LIN {X 0,Y 108.668,Z 991.691,A -85,B 0,C 180,E1 6722.041,E2 6722.041} C_VEL
LIN {X 0,Y 115.964,Z 986.125,A -85,B 0,C 180,E1 6711.629,E2 6711.629} C_VEL
LIN {X 0,Y 125.828,Z 978.975,A -85,B 0,C 180,E1 6703.029,E2 6703.029} C_VEL
LIN {X 0,Y 137.396,Z 970.37,A -85,B 0,C 180,E1 6696.117,E2 6696.117} C_VEL
LIN {X 0,Y 150.62,Z 959.785,A -85,B 0,C 180,E1 6690.352,E2 6690.352} C_VEL
LIN {X 0,Y 164.355,Z 947.613,A -85,B 0,C 180,E1 6685.798,E2 6685.798} C_VEL
LIN {X 0,Y 178.144,Z 933.873,A -85,B 0,C 180,E1 6682.172,E2 6682.172} C_VEL
LIN {X 0,Y 191.294,Z 919.026,A -85,B 0,C 180,E1 6679.367,E2 6679.367} C_VEL
LIN {X 0,Y 203.581,Z 903.149,A -85,B 0,C 180,E1 6677.161,E2 6677.161} C_VEL
LIN {X 0,Y 214.716,Z 886.544,A -85,B 0,C 180,E1 6675.442,E2 6675.442} C_VEL
LIN {X 0,Y 224.723,Z 869.138,A -85,B 0,C 180,E1 6674.088,E2 6674.088} C_VEL
LIN {X 0,Y 233.483,Z 851.076,A -85,B 0,C 180,E1 6673.039,E2 6673.039} C_VEL
LIN {X 0,Y 241.401,Z 830.942,A -85,B 0,C 180,E1 6672.186,E2 6672.186} C_VEL
LIN {X 0,Y 247.582,Z 810.659,A -85,B 0,C 180,E1 6671.567,E2 6671.567} C_VEL
LIN {X 0,Y 252.1,Z 790.058,A -85,B 0,C 180,E1 6671.085,E2 6671.085} C_VEL
LIN {X 0,Y 255.437,Z 766.946,A -85,B 0,C 180,E1 6670.837,E2 6670.837} C_VEL
LIN {X 0,Y 255.799,Z 763.582,A -85,B 0,C 180,E1 6670.771,E2 6670.771} C_VEL
LIN {X 0,Y 256.748,Z 736.616,A -85,B 0,C 180,E1 6667.524,E2 6667.524} C_VEL
LIN {X 0,Y 258.923,Z 706.753,A -85,B 0,C 180,E1 6664.457,E2 6664.457} C_VEL
LIN {X 0,Y 259.843,Z 696.602,A -85,B 0,C 180,E1 6663.474,E2 6663.474} C_VEL
LIN {X 0,Y 260.238,Z 689.281,A -85,B 0,C 180,E1 6660.825,E2 6660.825} C_VEL
LIN {X 0,Y 262.188,Z 677.578,A -85,B 0,C 180,E1 6656.009,E2 6656.009} C_VEL
LIN {X 0,Y 264.904,Z 669.637,A -85,B 0,C 180,E1 6652.19,E2 6652.19} C_VEL
LIN {X 0,Y 265.193,Z 670.053,A -85,B 0,C 180,E1 6651.653,E2 6651.653} C_VEL
LIN {X 0,Y 265.852,Z 672.18,A -85,B 0,C 180,E1 6650.356,E2 6650.356} C_VEL
LIN {X 0,Y 253.789,Z 778.906,A -85,B 0,C 180,E1 6648.472,E2 6648.472} C_VEL
LIN {X 0,Y 249.847,Z 799.249,A -85,B 0,C 180,E1 6647.946,E2 6647.946} C_VEL
LIN {X 0,Y 244.412,Z 819.077,A -85,B 0,C 180,E1 6647.237,E2 6647.237} C_VEL
LIN {X 0,Y 237.235,Z 839.076,A -85,B 0,C 180,E1 6646.276,E2 6646.276} C_VEL
LIN {X 0,Y 229.134,Z 857.25,A -85,B 0,C 180,E1 6645.133,E2 6645.133} C_VEL
LIN {X 0,Y 219.778,Z 874.734,A -85,B 0,C 180,E1 6643.719,E2 6643.719} C_VEL
LIN {X 0,Y 208.758,Z 892.029,A -85,B 0,C 180,E1 6641.89,E2 6641.89} C_VEL
LIN {X 0,Y 197.188,Z 907.581,A -85,B 0,C 180,E1 6639.724,E2 6639.724} C_VEL
LIN {X 0,Y 184.631,Z 922.268,A -85,B 0,C 180,E1 6637.014,E2 6637.014} C_VEL
LIN {X 0,Y 171.721,Z 935.505,A -85,B 0,C 180,E1 6633.721,E2 6633.721} C_VEL
LIN {X 0,Y 158.692,Z 947.341,A -85,B 0,C 180,E1 6629.672,E2 6629.672} C_VEL
LIN {X 0,Y 145.849,Z 957.776,A -85,B 0,C 180,E1 6624.663,E2 6624.663} C_VEL
LIN {X 0,Y 133.035,Z 967.156,A -85,B 0,C 180,E1 6618.075,E2 6618.075} C_VEL
LIN {X 0,Y 121.672,Z 974.814,A -85,B 0,C 180,E1 6609.862,E2 6609.862} C_VEL
LIN {X 0,Y 112.966,Z 980.439,A -85,B 0,C 180,E1 6600.295,E2 6600.295} C_VEL
LIN {X 0,Y 107.484,Z 984.062,A -85,B 0,C 180,E1 6590.023,E2 6590.023} C_VEL
LIN {X 0,Y 104.893,Z 986.058,A -85,B 0,C 180,E1 6579.323,E2 6579.323} C_VEL
LIN {X 0,Y 104.395,Z 986.656,A -85,B 0,C 180,E1 6569.997,E2 6569.997} C_VEL
LIN {X 0,Y 104.885,Z 986.083,A -85,B 0,C 180,E1 6560.671,E2 6560.671} C_VEL
LIN {X 0,Y 107.419,Z 984.152,A -85,B 0,C 180,E1 6550.072,E2 6550.072} C_VEL
LIN {X 0,Y 112.922,Z 980.53,A -85,B 0,C 180,E1 6539.685,E2 6539.685} C_VEL
LIN {X 0,Y 121.613,Z 974.922,A -85,B 0,C 180,E1 6530.109,E2 6530.109} C_VEL
LIN {X 0,Y 132.383,Z 967.681,A -85,B 0,C 180,E1 6522.238,E2 6522.238} C_VEL
LIN {X 0,Y 144.419,Z 958.957,A -85,B 0,C 180,E1 6515.898,E2 6515.898} C_VEL
LIN {X 0,Y 157.325,Z 948.621,A -85,B 0,C 180,E1 6510.697,E2 6510.697} C_VEL
LIN {X 0,Y 147.051,Z 951.529,A -85,B 0,C 180,E1 6506.23,E2 6506.23} C_VEL
LIN {X 0,Y 136.461,Z 954.568,A -85,B 0,C 180,E1 6499.698,E2 6499.698} C_VEL
LIN {X 0,Y 128.082,Z 957.332,A -85,B 0,C 180,E1 6491.711,E2 6491.711} C_VEL
LIN {X 0,Y 122.949,Z 959.82,A -85,B 0,C 180,E1 6483.264,E2 6483.264} C_VEL
LIN {X 0,Y 120.93,Z 962.742,A -85,B 0,C 180,E1 6471.921,E2 6471.921} C_VEL
LIN {X 0,Y 125.352,Z 965.819,A -85,B 0,C 180,E1 6458.475,E2 6458.475} C_VEL
LIN {X 0,Y 139.784,Z 968.622,A -85,B 0,C 180,E1 6445.025,E2 6445.025} C_VEL
LIN {X 0,Y 127.566,Z 977.809,A -85,B 0,C 180,E1 6438.129,E2 6438.129} C_VEL
LIN {X 0,Y 117.313,Z 985.24,A -85,B 0,C 180,E1 6429.738,E2 6429.738} C_VEL
LIN {X 0,Y 109.807,Z 990.867,A -85,B 0,C 180,E1 6420.021,E2 6420.021} C_VEL
LIN {X 0,Y 106.896,Z 992.481,A -85,B 0,C 180,E1 6416.302,E2 6416.302} C_VEL
LIN {X 0,Y 97.532,Z 995.483,A -85,B 0,C 180,E1 6405.695,E2 6405.695} C_VEL
LIN {X 0,Y 96.381,Z 996.081,A -85,B 0,C 180,E1 6401.813,E2 6401.813} C_VEL
LIN {X 0,Y 96.466,Z 996.89,A -85,B 0,C 180,E1 6392.974,E2 6392.974} C_VEL
LIN {X 0,Y 96.487,Z 996.912,A -85,B 0,C 180,E1 6387.628,E2 6387.628} C_VEL
LIN {X 0,Y 96.343,Z 996.122,A -85,B 0,C 180,E1 6378.631,E2 6378.631} C_VEL
LIN {X 0,Y 98.527,Z 993.582,A -85,B 0,C 180,E1 6366.689,E2 6366.689} C_VEL
LIN {X 0,Y 104.163,Z 989.385,A -85,B 0,C 180,E1 6355.508,E2 6355.508} C_VEL
LIN {X 0,Y 113.072,Z 983.454,A -85,B 0,C 180,E1 6345.691,E2 6345.691} C_VEL
LIN {X 0,Y 124.689,Z 975.635,A -85,B 0,C 180,E1 6337.456,E2 6337.456} C_VEL
LIN {X 0,Y 137.668,Z 966.274,A -85,B 0,C 180,E1 6331.021,E2 6331.021} C_VEL
LIN {X 0,Y 151.3,Z 955.493,A -85,B 0,C 180,E1 6326.01,E2 6326.01} C_VEL
LIN {X 0,Y 165.287,Z 943.149,A -85,B 0,C 180,E1 6322.027,E2 6322.027} C_VEL
LIN {X 0,Y 179.539,Z 928.903,A -85,B 0,C 180,E1 6318.79,E2 6318.79} C_VEL
LIN {X 0,Y 192.745,Z 913.813,A -85,B 0,C 180,E1 6316.331,E2 6316.331} C_VEL
LIN {X 0,Y 205.021,Z 897.675,A -85,B 0,C 180,E1 6314.401,E2 6314.401} C_VEL
LIN {X 0,Y 216.392,Z 880.245,A -85,B 0,C 180,E1 6312.859,E2 6312.859} C_VEL
LIN {X 0,Y 226.628,Z 861.559,A -85,B 0,C 180,E1 6311.646,E2 6311.646} C_VEL
LIN {X 0,Y 235.094,Z 842.869,A -85,B 0,C 180,E1 6310.758,E2 6310.758} C_VEL
LIN {X 0,Y 242.203,Z 823.431,A -85,B 0,C 180,E1 6310.085,E2 6310.085} C_VEL
LIN {X 0,Y 248.112,Z 802.126,A -85,B 0,C 180,E1 6309.543,E2 6309.543} C_VEL
LIN {X 0,Y 252.098,Z 781.253,A -85,B 0,C 180,E1 6309.166,E2 6309.166} C_VEL
LIN {X 0,Y 254.15,Z 765.555,A -85,B 0,C 180,E1 6309.011,E2 6309.011} C_VEL
LIN {X 0,Y 255.491,Z 739.464,A -85,B 0,C 180,E1 6305.868,E2 6305.868} C_VEL
LIN {X 0,Y 258.115,Z 709.106,A -85,B 0,C 180,E1 6302.761,E2 6302.761} C_VEL
LIN {X 0,Y 258.855,Z 701.864,A -85,B 0,C 180,E1 6302.047,E2 6302.047} C_VEL
LIN {X 0,Y 259.505,Z 694.909,A -85,B 0,C 180,E1 6299.448,E2 6299.448} C_VEL
LIN {X 0,Y 261.599,Z 684.612,A -85,B 0,C 180,E1 6295.176,E2 6295.176} C_VEL
LIN {X 0,Y 264.006,Z 677.964,A -85,B 0,C 180,E1 6291.973,E2 6291.973} C_VEL
LIN {X 0,Y 252.295,Z 779.354,A -85,B 0,C 180,E1 6290.249,E2 6290.249} C_VEL
LIN {X 0,Y 248.269,Z 799.753,A -85,B 0,C 180,E1 6289.747,E2 6289.747} C_VEL
LIN {X 0,Y 242.759,Z 819.493,A -85,B 0,C 180,E1 6289.078,E2 6289.078} C_VEL
LIN {X 0,Y 235.463,Z 839.469,A -85,B 0,C 180,E1 6288.17,E2 6288.17} C_VEL
LIN {X 0,Y 227.208,Z 857.649,A -85,B 0,C 180,E1 6287.088,E2 6287.088} C_VEL
LIN {X 0,Y 217.663,Z 875.137,A -85,B 0,C 180,E1 6285.749,E2 6285.749} C_VEL
LIN {X 0,Y 206.443,Z 892.371,A -85,B 0,C 180,E1 6284.021,E2 6284.021} C_VEL
LIN {X 0,Y 194.54,Z 907.991,A -85,B 0,C 180,E1 6281.952,E2 6281.952} C_VEL
LIN {X 0,Y 181.629,Z 922.681,A -85,B 0,C 180,E1 6279.36,E2 6279.36} C_VEL
LIN {X 0,Y 168.111,Z 936.089,A -85,B 0,C 180,E1 6276.143,E2 6276.143} C_VEL
LIN {X 0,Y 154.756,Z 947.757,A -85,B 0,C 180,E1 6272.265,E2 6272.265} C_VEL
LIN {X 0,Y 141.31,Z 958.194,A -85,B 0,C 180,E1 6267.348,E2 6267.348} C_VEL
LIN {X 0,Y 127.75,Z 967.574,A -85,B 0,C 180,E1 6260.787,E2 6260.787} C_VEL
LIN {X 0,Y 116.08,Z 974.902,A -85,B 0,C 180,E1 6252.877,E2 6252.877} C_VEL
LIN {X 0,Y 106.817,Z 980.371,A -85,B 0,C 180,E1 6243.519,E2 6243.519} C_VEL
LIN {X 0,Y 100.443,Z 984.148,A -85,B 0,C 180,E1 6232.841,E2 6232.841} C_VEL
LIN {X 0,Y 97.156,Z 986.346,A -85,B 0,C 180,E1 6221.273,E2 6221.273} C_VEL
LIN {X 0,Y 96.405,Z 987.005,A -85,B 0,C 180,E1 6211.78,E2 6211.78} C_VEL
LIN {X 0,Y 96.706,Z 986.749,A -85,B 0,C 180,E1 6202.272,E2 6202.272} C_VEL
LIN {X 0,Y 98.745,Z 985.269,A -85,B 0,C 180,E1 6191.703,E2 6191.703} C_VEL
LIN {X 0,Y 103.864,Z 982.144,A -85,B 0,C 180,E1 6180.593,E2 6180.593} C_VEL
LIN {X 0,Y 112.481,Z 977.086,A -85,B 0,C 180,E1 6170.204,E2 6170.204} C_VEL
LIN {X 0,Y 123.359,Z 970.453,A -85,B 0,C 180,E1 6161.778,E2 6161.778} C_VEL
LIN {X 0,Y 135.623,Z 962.37,A -85,B 0,C 180,E1 6155.078,E2 6155.078} C_VEL
LIN {X 0,Y 146.77,Z 954.193,A -85,B 0,C 180,E1 6150.387,E2 6150.387} C_VEL
LIN {X 0,Y 130.806,Z 958.339,A -85,B 0,C 180,E1 6141.526,E2 6141.526} C_VEL
LIN {X 0,Y 121.494,Z 961.15,A -85,B 0,C 180,E1 6132.839,E2 6132.839} C_VEL
LIN {X 0,Y 116.002,Z 963.516,A -85,B 0,C 180,E1 6123.955,E2 6123.955} C_VEL
LIN {X 0,Y 113.721,Z 966.225,A -85,B 0,C 180,E1 6112.422,E2 6112.422} C_VEL
LIN {X 0,Y 118.395,Z 969.376,A -85,B 0,C 180,E1 6097.665,E2 6097.665} C_VEL
LIN {X 0,Y 130.332,Z 971.766,A -85,B 0,C 180,E1 6085.562,E2 6085.562} C_VEL
LIN {X 0,Y 118.034,Z 980.243,A -85,B 0,C 180,E1 6078.201,E2 6078.201} C_VEL
LIN {X 0,Y 107.403,Z 987.311,A -85,B 0,C 180,E1 6068.593,E2 6068.593} C_VEL
LIN {X 0,Y 100.103,Z 992.425,A -85,B 0,C 180,E1 6057.259,E2 6057.259} C_VEL
LIN {X 0,Y 96.753,Z 995.452,A -85,B 0,C 180,E1 6045.59,E2 6045.59} C_VEL
LIN {X 0,Y 96.381,Z 996.081,A -85,B 0,C 180,E1 6041.813,E2 6041.813} C_VEL
LIN {X 0,Y 95.319,Z 996.58,A -85,B 0,C 180,E1 6037.558,E2 6037.558} C_VEL
LIN {X 0,Y 92.506,Z 996.742,A -85,B 0,C 180,E1 6032.007,E2 6032.007} C_VEL
LIN {X 0,Y 88.396,Z 996.199,A -85,B 0,C 180,E1 6021.798,E2 6021.798} C_VEL
LIN {X 0,Y 88.298,Z 995.978,A -85,B 0,C 180,E1 6019.947,E2 6019.947} C_VEL
LIN {X 0,Y 90.039,Z 994.007,A -85,B 0,C 180,E1 6007.821,E2 6007.821} C_VEL
LIN {X 0,Y 95.911,Z 989.964,A -85,B 0,C 180,E1 5995.019,E2 5995.019} C_VEL
LIN {X 0,Y 105.121,Z 984.331,A -85,B 0,C 180,E1 5984.495,E2 5984.495} C_VEL
LIN {X 0,Y 117.166,Z 976.876,A -85,B 0,C 180,E1 5975.84,E2 5975.84} C_VEL
LIN {X 0,Y 131.337,Z 967.426,A -85,B 0,C 180,E1 5968.902,E2 5968.902} C_VEL
LIN {X 0,Y 146.246,Z 956.361,A -85,B 0,C 180,E1 5963.638,E2 5963.638} C_VEL
LIN {X 0,Y 160.46,Z 944.482,A -85,B 0,C 180,E1 5959.801,E2 5959.801} C_VEL
LIN {X 0,Y 174.409,Z 931.286,A -85,B 0,C 180,E1 5956.793,E2 5956.793} C_VEL
LIN {X 0,Y 188.338,Z 916.157,A -85,B 0,C 180,E1 5954.342,E2 5954.342} C_VEL
LIN {X 0,Y 201.277,Z 899.839,A -85,B 0,C 180,E1 5952.434,E2 5952.434} C_VEL
LIN {X 0,Y 212.854,Z 882.789,A -85,B 0,C 180,E1 5950.969,E2 5950.969} C_VEL
LIN {X 0,Y 223.238,Z 864.744,A -85,B 0,C 180,E1 5949.825,E2 5949.825} C_VEL
LIN {X 0,Y 232.29,Z 845.836,A -85,B 0,C 180,E1 5948.949,E2 5948.949} C_VEL
LIN {X 0,Y 239.724,Z 826.696,A -85,B 0,C 180,E1 5948.303,E2 5948.303} C_VEL
LIN {X 0,Y 245.869,Z 806.184,A -85,B 0,C 180,E1 5947.797,E2 5947.797} C_VEL
LIN {X 0,Y 250.344,Z 784.986,A -85,B 0,C 180,E1 5947.404,E2 5947.404} C_VEL
LIN {X 0,Y 252.729,Z 767.652,A -85,B 0,C 180,E1 5947.23,E2 5947.23} C_VEL
LIN {X 0,Y 254.698,Z 739.448,A -85,B 0,C 180,E1 5943.883,E2 5943.883} C_VEL
LIN {X 0,Y 257.88,Z 708.454,A -85,B 0,C 180,E1 5940.777,E2 5940.777} C_VEL
LIN {X 0,Y 258.046,Z 706.967,A -85,B 0,C 180,E1 5940.555,E2 5940.555} C_VEL
LIN {X 0,Y 260.917,Z 692.086,A -85,B 0,C 180,E1 5934.557,E2 5934.557} C_VEL
LIN {X 0,Y 261.634,Z 690.138,A -85,B 0,C 180,E1 5933.511,E2 5933.511} C_VEL
LIN {X 0,Y 251.012,Z 780.054,A -85,B 0,C 180,E1 5932.04,E2 5932.04} C_VEL
LIN {X 0,Y 246.912,Z 800.368,A -85,B 0,C 180,E1 5931.566,E2 5931.566} C_VEL
LIN {X 0,Y 241.363,Z 819.898,A -85,B 0,C 180,E1 5930.943,E2 5930.943} C_VEL
LIN {X 0,Y 233.952,Z 839.861,A -85,B 0,C 180,E1 5930.091,E2 5930.091} C_VEL
LIN {X 0,Y 225.552,Z 858.049,A -85,B 0,C 180,E1 5929.074,E2 5929.074} C_VEL
LIN {X 0,Y 215.826,Z 875.541,A -85,B 0,C 180,E1 5927.817,E2 5927.817} C_VEL
LIN {X 0,Y 204.374,Z 892.778,A -85,B 0,C 180,E1 5926.19,E2 5926.19} C_VEL
LIN {X 0,Y 192.195,Z 908.402,A -85,B 0,C 180,E1 5924.238,E2 5924.238} C_VEL
LIN {X 0,Y 178.942,Z 923.093,A -85,B 0,C 180,E1 5921.781,E2 5921.781} C_VEL
LIN {X 0,Y 164.677,Z 936.795,A -85,B 0,C 180,E1 5918.635,E2 5918.635} C_VEL
LIN {X 0,Y 150.348,Z 948.793,A -85,B 0,C 180,E1 5914.743,E2 5914.743} C_VEL
LIN {X 0,Y 136.348,Z 959.111,A -85,B 0,C 180,E1 5909.913,E2 5909.913} C_VEL
LIN {X 0,Y 122.776,Z 967.992,A -85,B 0,C 180,E1 5903.725,E2 5903.725} C_VEL
LIN {X 0,Y 109.702,Z 975.651,A -85,B 0,C 180,E1 5895.306,E2 5895.306} C_VEL
LIN {X 0,Y 99.305,Z 981.275,A -85,B 0,C 180,E1 5885.019,E2 5885.019} C_VEL
LIN {X 0,Y 92.523,Z 984.866,A -85,B 0,C 180,E1 5873.565,E2 5873.565} C_VEL
LIN {X 0,Y 89.095,Z 986.885,A -85,B 0,C 180,E1 5860.995,E2 5860.995} C_VEL
LIN {X 0,Y 88.415,Z 987.479,A -85,B 0,C 180,E1 5849.997,E2 5849.997} C_VEL
LIN {X 0,Y 89.086,Z 986.91,A -85,B 0,C 180,E1 5838.997,E2 5838.997} C_VEL
LIN {X 0,Y 92.247,Z 985.074,A -85,B 0,C 180,E1 5827.029,E2 5827.029} C_VEL
LIN {X 0,Y 99.263,Z 981.362,A -85,B 0,C 180,E1 5814.956,E2 5814.956} C_VEL
LIN {X 0,Y 109.851,Z 975.646,A -85,B 0,C 180,E1 5804.496,E2 5804.496} C_VEL
LIN {X 0,Y 122.715,Z 968.129,A -85,B 0,C 180,E1 5796.227,E2 5796.227} C_VEL
LIN {X 0,Y 136.43,Z 959.178,A -85,B 0,C 180,E1 5789.952,E2 5789.952} C_VEL
LIN {X 0,Y 124.656,Z 961.988,A -85,B 0,C 180,E1 5783.144,E2 5783.144} C_VEL
LIN {X 0,Y 115.183,Z 964.621,A -85,B 0,C 180,E1 5774.581,E2 5774.581} C_VEL
LIN {X 0,Y 108.981,Z 967.029,A -85,B 0,C 180,E1 5764.737,E2 5764.737} C_VEL
LIN {X 0,Y 106.47,Z 969.602,A -85,B 0,C 180,E1 5752.446,E2 5752.446} C_VEL
LIN {X 0,Y 111.332,Z 972.629,A -85,B 0,C 180,E1 5736.725,E2 5736.725} C_VEL
LIN {X 0,Y 121.009,Z 974.573,A -85,B 0,C 180,E1 5726.251,E2 5726.251} C_VEL
LIN {X 0,Y 108.504,Z 982.374,A -85,B 0,C 180,E1 5718.285,E2 5718.285} C_VEL
LIN {X 0,Y 98.359,Z 988.484,A -85,B 0,C 180,E1 5708.326,E2 5708.326} C_VEL
LIN {X 0,Y 91.323,Z 993.026,A -85,B 0,C 180,E1 5695.976,E2 5695.976} C_VEL
LIN {X 0,Y 88.467,Z 995.643,A -85,B 0,C 180,E1 5683.068,E2 5683.068} C_VEL
LIN {X 0,Y 88.459,Z 996.477,A -85,B 0,C 180,E1 5673.243,E2 5673.243} C_VEL
LIN {X 0,Y 88.484,Z 996.499,A -85,B 0,C 180,E1 5667.413,E2 5667.413} C_VEL
LIN {X 0,Y 88.298,Z 995.978,A -85,B 0,C 180,E1 5659.947,E2 5659.947} C_VEL
LIN {X 0,Y 87.663,Z 995.347,A -85,B 0,C 180,E1 5654.929,E2 5654.929} C_VEL
LIN {X 0,Y 85.123,Z 993.386,A -85,B 0,C 180,E1 5644.717,E2 5644.717} C_VEL
LIN {X 0,Y 85.592,Z 991.753,A -85,B 0,C 180,E1 5638.425,E2 5638.425} C_VEL
LIN {X 0,Y 86.354,Z 991.183,A -85,B 0,C 180,E1 5636.672,E2 5636.672} C_VEL
LIN {X 0,Y 95.582,Z 986.11,A -85,B 0,C 180,E1 5624.661,E2 5624.661} C_VEL
LIN {X 0,Y 108.387,Z 978.945,A -85,B 0,C 180,E1 5614.818,E2 5614.818} C_VEL
LIN {X 0,Y 122.882,Z 970.112,A -85,B 0,C 180,E1 5607.518,E2 5607.518} C_VEL
LIN {X 0,Y 137.941,Z 959.823,A -85,B 0,C 180,E1 5602.142,E2 5602.142} C_VEL
LIN {X 0,Y 152.606,Z 948.48,A -85,B 0,C 180,E1 5598.197,E2 5598.197} C_VEL
LIN {X 0,Y 167.691,Z 935.177,A -85,B 0,C 180,E1 5595.006,E2 5595.006} C_VEL
LIN {X 0,Y 182.315,Z 920.329,A -85,B 0,C 180,E1 5592.535,E2 5592.535} C_VEL
LIN {X 0,Y 195.365,Z 905.022,A -85,B 0,C 180,E1 5590.7,E2 5590.7} C_VEL
LIN {X 0,Y 207.655,Z 888.259,A -85,B 0,C 180,E1 5589.231,E2 5589.231} C_VEL
LIN {X 0,Y 218.642,Z 870.536,A -85,B 0,C 180,E1 5588.093,E2 5588.093} C_VEL
LIN {X 0,Y 228.273,Z 851.881,A -85,B 0,C 180,E1 5587.221,E2 5587.221} C_VEL
LIN {X 0,Y 236.024,Z 833.581,A -85,B 0,C 180,E1 5586.596,E2 5586.596} C_VEL
LIN {X 0,Y 243.044,Z 812.513,A -85,B 0,C 180,E1 5586.075,E2 5586.075} C_VEL
LIN {X 0,Y 248.142,Z 791.369,A -85,B 0,C 180,E1 5585.668,E2 5585.668} C_VEL
LIN {X 0,Y 251.43,Z 770.926,A -85,B 0,C 180,E1 5585.483,E2 5585.483} C_VEL
LIN {X 0,Y 251.609,Z 768.944,A -85,B 0,C 180,E1 5585.329,E2 5585.329} C_VEL
LIN {X 0,Y 254.288,Z 738.743,A -85,B 0,C 180,E1 5581.83,E2 5581.83} C_VEL
LIN {X 0,Y 257.365,Z 712.416,A -85,B 0,C 180,E1 5579.165,E2 5579.165} C_VEL
LIN {X 0,Y 259.438,Z 702.446,A -85,B 0,C 180,E1 5575.073,E2 5575.073} C_VEL
LIN {X 0,Y 249.998,Z 780.612,A -85,B 0,C 180,E1 5573.851,E2 5573.851} C_VEL
LIN {X 0,Y 245.807,Z 800.988,A -85,B 0,C 180,E1 5573.403,E2 5573.403} C_VEL
LIN {X 0,Y 240.225,Z 820.305,A -85,B 0,C 180,E1 5572.827,E2 5572.827} C_VEL
LIN {X 0,Y 232.708,Z 840.253,A -85,B 0,C 180,E1 5572.034,E2 5572.034} C_VEL
LIN {X 0,Y 224.17,Z 858.447,A -85,B 0,C 180,E1 5571.087,E2 5571.087} C_VEL
LIN {X 0,Y 214.275,Z 875.944,A -85,B 0,C 180,E1 5569.917,E2 5569.917} C_VEL
LIN {X 0,Y 202.604,Z 893.185,A -85,B 0,C 180,E1 5568.401,E2 5568.401} C_VEL
LIN {X 0,Y 190.163,Z 908.811,A -85,B 0,C 180,E1 5566.577,E2 5566.577} C_VEL
LIN {X 0,Y 176.583,Z 923.506,A -85,B 0,C 180,E1 5564.27,E2 5564.27} C_VEL
LIN {X 0,Y 162.439,Z 936.748,A -85,B 0,C 180,E1 5561.421,E2 5561.421} C_VEL
LIN {X 0,Y 147.907,Z 948.59,A -85,B 0,C 180,E1 5557.833,E2 5557.833} C_VEL
LIN {X 0,Y 133.256,Z 959.028,A -85,B 0,C 180,E1 5553.234,E2 5553.234} C_VEL
LIN {X 0,Y 118.152,Z 968.41,A -85,B 0,C 180,E1 5546.902,E2 5546.902} C_VEL
LIN {X 0,Y 104.15,Z 976.069,A -85,B 0,C 180,E1 5538.483,E2 5538.483} C_VEL
LIN {X 0,Y 92.782,Z 981.693,A -85,B 0,C 180,E1 5527.894,E2 5527.894} C_VEL
LIN {X 0,Y 85.179,Z 985.282,A -85,B 0,C 180,E1 5515.738,E2 5515.738} C_VEL
LIN {X 0,Y 81.228,Z 987.299,A -85,B 0,C 180,E1 5502.075,E2 5502.075} C_VEL
LIN {X 0,Y 80.425,Z 987.89,A -85,B 0,C 180,E1 5489.996,E2 5489.996} C_VEL
LIN {X 0,Y 81.22,Z 987.323,A -85,B 0,C 180,E1 5477.916,E2 5477.916} C_VEL
LIN {X 0,Y 84.868,Z 985.49,A -85,B 0,C 180,E1 5464.9,E2 5464.9} C_VEL
LIN {X 0,Y 92.74,Z 981.779,A -85,B 0,C 180,E1 5452.078,E2 5452.078} C_VEL
LIN {X 0,Y 104.097,Z 976.172,A -85,B 0,C 180,E1 5441.475,E2 5441.475} C_VEL
LIN {X 0,Y 117.379,Z 968.936,A -85,B 0,C 180,E1 5433.402,E2 5433.402} C_VEL
LIN {X 0,Y 125.897,Z 963.88,A -85,B 0,C 180,E1 5429.499,E2 5429.499} C_VEL
LIN {X 0,Y 109.281,Z 967.732,A -85,B 0,C 180,E1 5417.025,E2 5417.025} C_VEL
LIN {X 0,Y 101.86,Z 970.281,A -85,B 0,C 180,E1 5405.634,E2 5405.634} C_VEL
LIN {X 0,Y 99.133,Z 972.793,A -85,B 0,C 180,E1 5392.467,E2 5392.467} C_VEL
LIN {X 0,Y 104.22,Z 975.673,A -85,B 0,C 180,E1 5375.637,E2 5375.637} C_VEL
LIN {X 0,Y 111.613,Z 977.111,A -85,B 0,C 180,E1 5367.02,E2 5367.02} C_VEL
LIN {X 0,Y 98.372,Z 984.613,A -85,B 0,C 180,E1 5357.87,E2 5357.87} C_VEL
LIN {X 0,Y 88.09,Z 990.241,A -85,B 0,C 180,E1 5346.177,E2 5346.177} C_VEL
LIN {X 0,Y 82.136,Z 993.87,A -85,B 0,C 180,E1 5332.93,E2 5332.93} C_VEL
LIN {X 0,Y 80.308,Z 995.761,A -85,B 0,C 180,E1 5319.318,E2 5319.318} C_VEL
LIN {X 0,Y 80.588,Z 996.183,A -85,B 0,C 180,E1 5310.004,E2 5310.004} C_VEL
LIN {X 0,Y 80.292,Z 995.745,A -85,B 0,C 180,E1 5300.687,E2 5300.687} C_VEL
LIN {X 0,Y 82.113,Z 993.843,A -85,B 0,C 180,E1 5287.071,E2 5287.071} C_VEL
LIN {X 0,Y 86.354,Z 991.183,A -85,B 0,C 180,E1 5276.672,E2 5276.672} C_VEL
LIN {X 0,Y 88.288,Z 989.594,A -85,B 0,C 180,E1 5271.849,E2 5271.849} C_VEL
LIN {X 0,Y 92.995,Z 984.521,A -85,B 0,C 180,E1 5259.103,E2 5259.103} C_VEL
LIN {X 0,Y 96.329,Z 982.492,A -85,B 0,C 180,E1 5255.831,E2 5255.831} C_VEL
LIN {X 0,Y 111.39,Z 974.362,A -85,B 0,C 180,E1 5247.303,E2 5247.303} C_VEL
LIN {X 0,Y 126.716,Z 965.004,A -85,B 0,C 180,E1 5241.402,E2 5241.402} C_VEL
LIN {X 0,Y 142.227,Z 954.227,A -85,B 0,C 180,E1 5237.051,E2 5237.051} C_VEL
LIN {X 0,Y 157.492,Z 942.084,A -85,B 0,C 180,E1 5233.759,E2 5233.759} C_VEL
LIN {X 0,Y 172.271,Z 928.585,A -85,B 0,C 180,E1 5231.233,E2 5231.233} C_VEL
LIN {X 0,Y 186.403,Z 913.679,A -85,B 0,C 180,E1 5229.26,E2 5229.26} C_VEL
LIN {X 0,Y 199.769,Z 897.261,A -85,B 0,C 180,E1 5227.702,E2 5227.702} C_VEL
LIN {X 0,Y 211.752,Z 879.886,A -85,B 0,C 180,E1 5226.507,E2 5226.507} C_VEL
LIN {X 0,Y 222.03,Z 862.147,A -85,B 0,C 180,E1 5225.618,E2 5225.618} C_VEL
LIN {X 0,Y 230.823,Z 843.924,A -85,B 0,C 180,E1 5224.951,E2 5224.951} C_VEL
LIN {X 0,Y 238.671,Z 823.735,A -85,B 0,C 180,E1 5224.421,E2 5224.421} C_VEL
LIN {X 0,Y 244.701,Z 803.397,A -85,B 0,C 180,E1 5224.024,E2 5224.024} C_VEL
LIN {X 0,Y 248.943,Z 783.329,A -85,B 0,C 180,E1 5223.732,E2 5223.732} C_VEL
LIN {X 0,Y 250.633,Z 771.769,A -85,B 0,C 180,E1 5223.616,E2 5223.616} C_VEL
LIN {X 0,Y 253.764,Z 741.686,A -85,B 0,C 180,E1 5220.155,E2 5220.155} C_VEL
LIN {X 0,Y 256.818,Z 718.012,A -85,B 0,C 180,E1 5217.768,E2 5217.768} C_VEL
LIN {X 0,Y 257.353,Z 715.466,A -85,B 0,C 180,E1 5216.651,E2 5216.651} C_VEL
LIN {X 0,Y 249.196,Z 781.427,A -85,B 0,C 180,E1 5215.67,E2 5215.67} C_VEL
LIN {X 0,Y 244.871,Z 801.964,A -85,B 0,C 180,E1 5215.246,E2 5215.246} C_VEL
LIN {X 0,Y 238.986,Z 821.798,A -85,B 0,C 180,E1 5214.691,E2 5214.691} C_VEL
LIN {X 0,Y 231.251,Z 841.752,A -85,B 0,C 180,E1 5213.948,E2 5213.948} C_VEL
LIN {X 0,Y 222.027,Z 860.761,A -85,B 0,C 180,E1 5213.016,E2 5213.016} C_VEL
LIN {X 0,Y 211.584,Z 878.522,A -85,B 0,C 180,E1 5211.885,E2 5211.885} C_VEL
LIN {X 0,Y 200.022,Z 895.097,A -85,B 0,C 180,E1 5210.505,E2 5210.505} C_VEL
LIN {X 0,Y 186.593,Z 911.396,A -85,B 0,C 180,E1 5208.689,E2 5208.689} C_VEL
LIN {X 0,Y 172.735,Z 925.732,A -85,B 0,C 180,E1 5206.512,E2 5206.512} C_VEL
LIN {X 0,Y 158.255,Z 938.669,A -85,B 0,C 180,E1 5203.803,E2 5203.803} C_VEL
LIN {X 0,Y 143.314,Z 950.245,A -85,B 0,C 180,E1 5200.359,E2 5200.359} C_VEL
LIN {X 0,Y 128.157,Z 960.446,A -85,B 0,C 180,E1 5195.891,E2 5195.891} C_VEL
LIN {X 0,Y 113.161,Z 969.22,A -85,B 0,C 180,E1 5189.98,E2 5189.98} C_VEL
LIN {X 0,Y 98.702,Z 976.603,A -85,B 0,C 180,E1 5181.833,E2 5181.833} C_VEL
LIN {X 0,Y 86.527,Z 982.111,A -85,B 0,C 180,E1 5171.193,E2 5171.193} C_VEL
LIN {X 0,Y 77.979,Z 985.699,A -85,B 0,C 180,E1 5158.317,E2 5158.317} C_VEL
LIN {X 0,Y 73.394,Z 987.712,A -85,B 0,C 180,E1 5143.387,E2 5143.387} C_VEL
LIN {X 0,Y 72.432,Z 988.283,A -85,B 0,C 180,E1 5130.787,E2 5130.787} C_VEL
LIN {X 0,Y 73.15,Z 987.861,A -85,B 0,C 180,E1 5118.164,E2 5118.164} C_VEL
LIN {X 0,Y 77.006,Z 986.195,A -85,B 0,C 180,E1 5103.799,E2 5103.799} C_VEL
LIN {X 0,Y 85.471,Z 982.609,A -85,B 0,C 180,E1 5089.949,E2 5089.949} C_VEL
LIN {X 0,Y 96.949,Z 977.462,A -85,B 0,C 180,E1 5079.327,E2 5079.327} C_VEL
LIN {X 0,Y 110.859,Z 970.526,A -85,B 0,C 180,E1 5071.033,E2 5071.033} C_VEL
LIN {X 0,Y 115.275,Z 968.146,A -85,B 0,C 180,E1 5068.893,E2 5068.893} C_VEL
LIN {X 0,Y 101.801,Z 971.069,A -85,B 0,C 180,E1 5057.727,E2 5057.727} C_VEL
LIN {X 0,Y 94.881,Z 973.189,A -85,B 0,C 180,E1 5047.266,E2 5047.266} C_VEL
LIN {X 0,Y 91.734,Z 975.802,A -85,B 0,C 180,E1 5031.855,E2 5031.855} C_VEL
LIN {X 0,Y 97.083,Z 978.526,A -85,B 0,C 180,E1 5014.371,E2 5014.371} C_VEL
LIN {X 0,Y 102.224,Z 979.477,A -85,B 0,C 180,E1 5007.924,E2 5007.924} C_VEL
LIN {X 0,Y 89.427,Z 986.042,A -85,B 0,C 180,E1 4998.518,E2 4998.518} C_VEL
LIN {X 0,Y 79.067,Z 991.127,A -85,B 0,C 180,E1 4985.575,E2 4985.575} C_VEL
LIN {X 0,Y 73.49,Z 994.194,A -85,B 0,C 180,E1 4970.721,E2 4970.721} C_VEL
LIN {X 0,Y 72.361,Z 995.584,A -85,B 0,C 180,E1 4955.821,E2 4955.821} C_VEL
LIN {X 0,Y 72.537,Z 995.726,A -85,B 0,C 180,E1 4948.424,E2 4948.424} C_VEL
LIN {X 0,Y 72.475,Z 995.021,A -85,B 0,C 180,E1 4936.44,E2 4936.44} C_VEL
LIN {X 0,Y 75.965,Z 992.656,A -85,B 0,C 180,E1 4920.861,E2 4920.861} C_VEL
LIN {X 0,Y 83.947,Z 988.644,A -85,B 0,C 180,E1 4907.247,E2 4907.247} C_VEL
LIN {X 0,Y 96.329,Z 982.492,A -85,B 0,C 180,E1 4895.831,E2 4895.831} C_VEL
LIN {X 0,Y 100.431,Z 979.975,A -85,B 0,C 180,E1 4892.284,E2 4892.284} C_VEL
LIN {X 0,Y 110.408,Z 972.731,A -85,B 0,C 180,E1 4882.87,E2 4882.87} C_VEL
LIN {X 0,Y 114.863,Z 969.999,A -85,B 0,C 180,E1 4880.749,E2 4880.749} C_VEL
LIN {X 0,Y 131.018,Z 960.023,A -85,B 0,C 180,E1 4875.945,E2 4875.945} C_VEL
LIN {X 0,Y 147.379,Z 948.347,A -85,B 0,C 180,E1 4872.339,E2 4872.339} C_VEL
LIN {X 0,Y 163.272,Z 935.193,A -85,B 0,C 180,E1 4869.628,E2 4869.628} C_VEL
LIN {X 0,Y 178.043,Z 921.027,A -85,B 0,C 180,E1 4867.623,E2 4867.623} C_VEL
LIN {X 0,Y 192.038,Z 905.416,A -85,B 0,C 180,E1 4866.052,E2 4866.052} C_VEL
LIN {X 0,Y 205.189,Z 888.161,A -85,B 0,C 180,E1 4864.811,E2 4864.811} C_VEL
LIN {X 0,Y 216.465,Z 870.536,A -85,B 0,C 180,E1 4863.899,E2 4863.899} C_VEL
LIN {X 0,Y 226.318,Z 852.083,A -85,B 0,C 180,E1 4863.209,E2 4863.209} C_VEL
LIN {X 0,Y 234.549,Z 833.244,A -85,B 0,C 180,E1 4862.703,E2 4862.703} C_VEL
LIN {X 0,Y 241.593,Z 812.72,A -85,B 0,C 180,E1 4862.305,E2 4862.305} C_VEL
LIN {X 0,Y 246.764,Z 792.244,A -85,B 0,C 180,E1 4861.982,E2 4861.982} C_VEL
LIN {X 0,Y 249.936,Z 773.78,A -85,B 0,C 180,E1 4861.791,E2 4861.791} C_VEL
LIN {X 0,Y 253.497,Z 744.346,A -85,B 0,C 180,E1 4858.446,E2 4858.446} C_VEL
LIN {X 0,Y 253.932,Z 741.148,A -85,B 0,C 180,E1 4858.079,E2 4858.079} C_VEL
LIN {X 0,Y 248.527,Z 782.97,A -85,B 0,C 180,E1 4857.486,E2 4857.486} C_VEL
LIN {X 0,Y 243.873,Z 804.255,A -85,B 0,C 180,E1 4857.071,E2 4857.071} C_VEL
LIN {X 0,Y 237.644,Z 824.351,A -85,B 0,C 180,E1 4856.541,E2 4856.541} C_VEL
LIN {X 0,Y 229.926,Z 843.547,A -85,B 0,C 180,E1 4855.873,E2 4855.873} C_VEL
LIN {X 0,Y 220.79,Z 861.896,A -85,B 0,C 180,E1 4855.04,E2 4855.04} C_VEL
LIN {X 0,Y 209.983,Z 879.846,A -85,B 0,C 180,E1 4853.986,E2 4853.986} C_VEL
LIN {X 0,Y 198.07,Z 896.477,A -85,B 0,C 180,E1 4852.704,E2 4852.704} C_VEL
LIN {X 0,Y 184.706,Z 912.322,A -85,B 0,C 180,E1 4851.074,E2 4851.074} C_VEL
LIN {X 0,Y 170.097,Z 927.052,A -85,B 0,C 180,E1 4848.998,E2 4848.998} C_VEL
LIN {X 0,Y 155.275,Z 939.836,A -85,B 0,C 180,E1 4846.483,E2 4846.483} C_VEL
LIN {X 0,Y 139.906,Z 951.28,A -85,B 0,C 180,E1 4843.259,E2 4843.259} C_VEL
LIN {X 0,Y 123.356,Z 961.863,A -85,B 0,C 180,E1 4838.762,E2 4838.762} C_VEL
LIN {X 0,Y 107.493,Z 970.54,A -85,B 0,C 180,E1 4832.884,E2 4832.884} C_VEL
LIN {X 0,Y 92.76,Z 977.492,A -85,B 0,C 180,E1 4825,E2 4825} C_VEL
LIN {X 0,Y 80.034,Z 982.759,A -85,B 0,C 180,E1 4814.39,E2 4814.39} C_VEL
LIN {X 0,Y 70.227,Z 986.416,A -85,B 0,C 180,E1 4799.883,E2 4799.883} C_VEL
LIN {X 0,Y 65.458,Z 988.188,A -85,B 0,C 180,E1 4784.141,E2 4784.141} C_VEL
LIN {X 0,Y 64.447,Z 988.713,A -85,B 0,C 180,E1 4769.995,E2 4769.995} C_VEL
LIN {X 0,Y 65.449,Z 988.212,A -85,B 0,C 180,E1 4755.847,E2 4755.847} C_VEL
LIN {X 0,Y 70.2,Z 986.471,A -85,B 0,C 180,E1 4740.094,E2 4740.094} C_VEL
LIN {X 0,Y 79.995,Z 982.83,A -85,B 0,C 180,E1 4725.572,E2 4725.572} C_VEL
LIN {X 0,Y 93.417,Z 977.296,A -85,B 0,C 180,E1 4714.493,E2 4714.493} C_VEL
LIN {X 0,Y 104.818,Z 971.972,A -85,B 0,C 180,E1 4708.208,E2 4708.208} C_VEL
LIN {X 0,Y 88.201,Z 975.823,A -85,B 0,C 180,E1 4689.791,E2 4689.791} C_VEL
LIN {X 0,Y 84.191,Z 978.467,A -85,B 0,C 180,E1 4671.808,E2 4671.808} C_VEL
LIN {X 0,Y 90.068,Z 981.147,A -85,B 0,C 180,E1 4652.641,E2 4652.641} C_VEL
LIN {X 0,Y 92.749,Z 981.666,A -85,B 0,C 180,E1 4648.947,E2 4648.947} C_VEL
LIN {X 0,Y 79.203,Z 987.783,A -85,B 0,C 180,E1 4638.006,E2 4638.006} C_VEL
LIN {X 0,Y 69.669,Z 991.933,A -85,B 0,C 180,E1 4624.041,E2 4624.041} C_VEL
LIN {X 0,Y 64.715,Z 994.542,A -85,B 0,C 180,E1 4606.152,E2 4606.152} C_VEL
LIN {X 0,Y 64.495,Z 995.292,A -85,B 0,C 180,E1 4592.67,E2 4592.67} C_VEL
LIN {X 0,Y 64.452,Z 995.26,A -85,B 0,C 180,E1 4586.447,E2 4586.447} C_VEL
LIN {X 0,Y 64.91,Z 994.369,A -85,B 0,C 180,E1 4572.062,E2 4572.062} C_VEL
LIN {X 0,Y 70.013,Z 991.722,A -85,B 0,C 180,E1 4555.168,E2 4555.168} C_VEL
LIN {X 0,Y 80.43,Z 987.157,A -85,B 0,C 180,E1 4540.69,E2 4540.69} C_VEL
LIN {X 0,Y 93.842,Z 981.024,A -85,B 0,C 180,E1 4530.347,E2 4530.347} C_VEL
LIN {X 0,Y 108.675,Z 973.49,A -85,B 0,C 180,E1 4523.074,E2 4523.074} C_VEL
LIN {X 0,Y 114.863,Z 969.999,A -85,B 0,C 180,E1 4520.749,E2 4520.749} C_VEL
LIN {X 0,Y 120.114,Z 966.747,A -85,B 0,C 180,E1 4518.451,E2 4518.451} C_VEL
LIN {X 0,Y 132.748,Z 957.368,A -85,B 0,C 180,E1 4511.989,E2 4511.989} C_VEL
LIN {X 0,Y 137.546,Z 953.906,A -85,B 0,C 180,E1 4510.676,E2 4510.676} C_VEL
LIN {X 0,Y 154.417,Z 941.244,A -85,B 0,C 180,E1 4507.841,E2 4507.841} C_VEL
LIN {X 0,Y 169.846,Z 927.75,A -85,B 0,C 180,E1 4505.82,E2 4505.82} C_VEL
LIN {X 0,Y 184.479,Z 912.856,A -85,B 0,C 180,E1 4504.263,E2 4504.263} C_VEL
LIN {X 0,Y 198.247,Z 896.44,A -85,B 0,C 180,E1 4503.048,E2 4503.048} C_VEL
LIN {X 0,Y 210.609,Z 878.96,A -85,B 0,C 180,E1 4502.121,E2 4502.121} C_VEL
LIN {X 0,Y 221.034,Z 861.344,A -85,B 0,C 180,E1 4501.451,E2 4501.451} C_VEL
LIN {X 0,Y 229.994,Z 843.137,A -85,B 0,C 180,E1 4500.951,E2 4500.951} C_VEL
LIN {X 0,Y 237.972,Z 822.969,A -85,B 0,C 180,E1 4500.561,E2 4500.561} C_VEL
LIN {X 0,Y 244.11,Z 802.627,A -85,B 0,C 180,E1 4500.259,E2 4500.259} C_VEL
LIN {X 0,Y 248.428,Z 782.583,A -85,B 0,C 180,E1 4500.042,E2 4500.042} C_VEL
LIN {X 0,Y 249.464,Z 775.759,A -85,B 0,C 180,E1 4499.957,E2 4499.957} C_VEL
LIN {X 0,Y 250.021,Z 772.054,A -85,B 0,C 180,E1 4499.488,E2 4499.488} C_VEL
LIN {X 0,Y 246.226,Z 793.811,A -85,B 0,C 180,E1 4499.159,E2 4499.159} C_VEL
LIN {X 0,Y 240.676,Z 814.671,A -85,B 0,C 180,E1 4498.729,E2 4498.729} C_VEL
LIN {X 0,Y 234.074,Z 833.181,A -85,B 0,C 180,E1 4498.223,E2 4498.223} C_VEL
LIN {X 0,Y 225.667,Z 851.975,A -85,B 0,C 180,E1 4497.561,E2 4497.561} C_VEL
LIN {X 0,Y 215.812,Z 869.99,A -85,B 0,C 180,E1 4496.745,E2 4496.745} C_VEL
LIN {X 0,Y 204.533,Z 887.194,A -85,B 0,C 180,E1 4495.732,E2 4495.732} C_VEL
LIN {X 0,Y 191.374,Z 904.04,A -85,B 0,C 180,E1 4494.421,E2 4494.421} C_VEL
LIN {X 0,Y 176.883,Z 919.692,A -85,B 0,C 180,E1 4492.753,E2 4492.753} C_VEL
LIN {X 0,Y 162.08,Z 933.302,A -85,B 0,C 180,E1 4490.749,E2 4490.749} C_VEL
LIN {X 0,Y 146.49,Z 945.603,A -85,B 0,C 180,E1 4488.184,E2 4488.184} C_VEL
LIN {X 0,Y 129.593,Z 956.981,A -85,B 0,C 180,E1 4484.662,E2 4484.662} C_VEL
LIN {X 0,Y 112.788,Z 966.573,A -85,B 0,C 180,E1 4479.99,E2 4479.99} C_VEL
LIN {X 0,Y 96.925,Z 974.27,A -85,B 0,C 180,E1 4473.82,E2 4473.82} C_VEL
LIN {X 0,Y 81.546,Z 980.602,A -85,B 0,C 180,E1 4464.809,E2 4464.809} C_VEL
LIN {X 0,Y 68.096,Z 985.326,A -85,B 0,C 180,E1 4451.35,E2 4451.35} C_VEL
LIN {X 0,Y 59.51,Z 988.045,A -85,B 0,C 180,E1 4433.775,E2 4433.775} C_VEL
LIN {X 0,Y 56.588,Z 989.002,A -85,B 0,C 180,E1 4416.08,E2 4416.08} C_VEL
LIN {X 0,Y 56.584,Z 989.01,A -85,B 0,C 180,E1 4403.908,E2 4403.908} C_VEL
LIN {X 0,Y 59.489,Z 988.084,A -85,B 0,C 180,E1 4386.205,E2 4386.205} C_VEL
LIN {X 0,Y 68.062,Z 985.384,A -85,B 0,C 180,E1 4368.613,E2 4368.613} C_VEL
LIN {X 0,Y 81.214,Z 980.782,A -85,B 0,C 180,E1 4355.356,E2 4355.356} C_VEL
LIN {X 0,Y 94.048,Z 975.572,A -85,B 0,C 180,E1 4347.379,E2 4347.379} C_VEL
LIN {X 0,Y 80.153,Z 978.676,A -85,B 0,C 180,E1 4329.334,E2 4329.334} C_VEL
LIN {X 0,Y 76.536,Z 980.859,A -85,B 0,C 180,E1 4312.495,E2 4312.495} C_VEL
LIN {X 0,Y 83.159,Z 983.513,A -85,B 0,C 180,E1 4290.466,E2 4290.466} C_VEL
LIN {X 0,Y 83.091,Z 983.647,A -85,B 0,C 180,E1 4290.05,E2 4290.05} C_VEL
LIN {X 0,Y 69.123,Z 989.19,A -85,B 0,C 180,E1 4277.544,E2 4277.544} C_VEL
LIN {X 0,Y 59.631,Z 992.856,A -85,B 0,C 180,E1 4260.206,E2 4260.206} C_VEL
LIN {X 0,Y 56.364,Z 994.64,A -85,B 0,C 180,E1 4241.258,E2 4241.258} C_VEL
LIN {X 0,Y 56.606,Z 994.948,A -85,B 0,C 180,E1 4230.005,E2 4230.005} C_VEL
LIN {X 0,Y 56.509,Z 994.415,A -85,B 0,C 180,E1 4215.663,E2 4215.663} C_VEL
LIN {X 0,Y 60.98,Z 992.319,A -85,B 0,C 180,E1 4196.125,E2 4196.125} C_VEL
LIN {X 0,Y 71.475,Z 988.268,A -85,B 0,C 180,E1 4179.707,E2 4179.707} C_VEL
LIN {X 0,Y 85.308,Z 982.631,A -85,B 0,C 180,E1 4168.481,E2 4168.481} C_VEL
LIN {X 0,Y 101.441,Z 975.178,A -85,B 0,C 180,E1 4160.557,E2 4160.557} C_VEL
LIN {X 0,Y 118.063,Z 966.257,A -85,B 0,C 180,E1 4155.115,E2 4155.115} C_VEL
LIN {X 0,Y 134.566,Z 955.963,A -85,B 0,C 180,E1 4151.259,E2 4151.259} C_VEL
LIN {X 0,Y 137.546,Z 953.906,A -85,B 0,C 180,E1 4150.676,E2 4150.676} C_VEL
LIN {X 0,Y 143.119,Z 949.824,A -85,B 0,C 180,E1 4149.228,E2 4149.228} C_VEL
LIN {X 0,Y 155.894,Z 939.1,A -85,B 0,C 180,E1 4144.907,E2 4144.907} C_VEL
LIN {X 0,Y 161.35,Z 934.352,A -85,B 0,C 180,E1 4143.894,E2 4143.894} C_VEL
LIN {X 0,Y 176.565,Z 920.252,A -85,B 0,C 180,E1 4142.377,E2 4142.377} C_VEL
LIN {X 0,Y 191.009,Z 904.591,A -85,B 0,C 180,E1 4141.197,E2 4141.197} C_VEL
LIN {X 0,Y 204.472,Z 887.338,A -85,B 0,C 180,E1 4140.28,E2 4140.28} C_VEL
LIN {X 0,Y 216.47,Z 868.919,A -85,B 0,C 180,E1 4139.59,E2 4139.59} C_VEL
LIN {X 0,Y 221.593,Z 859.841,A -85,B 0,C 180,E1 4139.32,E2 4139.32} C_VEL
LIN {X 0,Y 210.627,Z 878.16,A -85,B 0,C 180,E1 4138.504,E2 4138.504} C_VEL
LIN {X 0,Y 198.157,Z 895.468,A -85,B 0,C 180,E1 4137.486,E2 4137.486} C_VEL
LIN {X 0,Y 184.37,Z 911.54,A -85,B 0,C 180,E1 4136.22,E2 4136.22} C_VEL
LIN {X 0,Y 169.71,Z 926.063,A -85,B 0,C 180,E1 4134.652,E2 4134.652} C_VEL
LIN {X 0,Y 154.229,Z 939.158,A -85,B 0,C 180,E1 4132.683,E2 4132.683} C_VEL
LIN {X 0,Y 137.067,Z 951.493,A -85,B 0,C 180,E1 4129.977,E2 4129.977} C_VEL
LIN {X 0,Y 120.283,Z 961.698,A -85,B 0,C 180,E1 4126.537,E2 4126.537} C_VEL
LIN {X 0,Y 103.151,Z 970.475,A -85,B 0,C 180,E1 4121.783,E2 4121.783} C_VEL
LIN {X 0,Y 86.123,Z 977.743,A -85,B 0,C 180,E1 4114.89,E2 4114.89} C_VEL
LIN {X 0,Y 70.074,Z 983.365,A -85,B 0,C 180,E1 4104.414,E2 4104.414} C_VEL
LIN {X 0,Y 57.784,Z 986.949,A -85,B 0,C 180,E1 4089.802,E2 4089.802} C_VEL
LIN {X 0,Y 50.256,Z 988.954,A -85,B 0,C 180,E1 4069.762,E2 4069.762} C_VEL
LIN {X 0,Y 48.465,Z 989.518,A -85,B 0,C 180,E1 4051.176,E2 4051.176} C_VEL
LIN {X 0,Y 49.817,Z 989.101,A -85,B 0,C 180,E1 4032.472,E2 4032.472} C_VEL
LIN {X 0,Y 56.28,Z 987.443,A -85,B 0,C 180,E1 4012.833,E2 4012.833} C_VEL
LIN {X 0,Y 68.654,Z 983.859,A -85,B 0,C 180,E1 3996.766,E2 3996.766} C_VEL
LIN {X 0,Y 83.531,Z 978.747,A -85,B 0,C 180,E1 3986.29,E2 3986.29} C_VEL
LIN {X 0,Y 68.862,Z 982.776,A -85,B 0,C 180,E1 3955.838,E2 3955.838} C_VEL
LIN {X 0,Y 73.821,Z 985.305,A -85,B 0,C 180,E1 3931.698,E2 3931.698} C_VEL
LIN {X 0,Y 59.845,Z 990.142,A -85,B 0,C 180,E1 3918.066,E2 3918.066} C_VEL
LIN {X 0,Y 50.687,Z 993.181,A -85,B 0,C 180,E1 3898.264,E2 3898.264} C_VEL
LIN {X 0,Y 48.356,Z 994.38,A -85,B 0,C 180,E1 3877.039,E2 3877.039} C_VEL
LIN {X 0,Y 48.556,Z 994.514,A -85,B 0,C 180,E1 3868.826,E2 3868.826} C_VEL
LIN {X 0,Y 49.084,Z 993.764,A -85,B 0,C 180,E1 3849.746,E2 3849.746} C_VEL
LIN {X 0,Y 56.267,Z 991.217,A -85,B 0,C 180,E1 3827.534,E2 3827.534} C_VEL
LIN {X 0,Y 68.624,Z 987.105,A -85,B 0,C 180,E1 3812.329,E2 3812.329} C_VEL
LIN {X 0,Y 84.172,Z 981.258,A -85,B 0,C 180,E1 3802.108,E2 3802.108} C_VEL
LIN {X 0,Y 101.53,Z 973.505,A -85,B 0,C 180,E1 3795.194,E2 3795.194} C_VEL
LIN {X 0,Y 118.992,Z 964.259,A -85,B 0,C 180,E1 3790.557,E2 3790.557} C_VEL
LIN {X 0,Y 136.082,Z 953.607,A -85,B 0,C 180,E1 3787.311,E2 3787.311} C_VEL
LIN {X 0,Y 153.514,Z 940.824,A -85,B 0,C 180,E1 3784.811,E2 3784.811} C_VEL
LIN {X 0,Y 161.35,Z 934.352,A -85,B 0,C 180,E1 3783.894,E2 3783.894} C_VEL
LIN {X 0,Y 166.782,Z 929.528,A -85,B 0,C 180,E1 3782.963,E2 3782.963} C_VEL
LIN {X 0,Y 179.41,Z 916.959,A -85,B 0,C 180,E1 3779.837,E2 3779.837} C_VEL
LIN {X 0,Y 184.473,Z 911.489,A -85,B 0,C 180,E1 3779.17,E2 3779.17} C_VEL
LIN {X 0,Y 187.222,Z 908.438,A -85,B 0,C 180,E1 3778.991,E2 3778.991} C_VEL
LIN {X 0,Y 173.103,Z 922.844,A -85,B 0,C 180,E1 3777.755,E2 3777.755} C_VEL
LIN {X 0,Y 157.331,Z 936.559,A -85,B 0,C 180,E1 3776.132,E2 3776.132} C_VEL
LIN {X 0,Y 140.736,Z 948.768,A -85,B 0,C 180,E1 3774.04,E2 3774.04} C_VEL
LIN {X 0,Y 123.41,Z 959.49,A -85,B 0,C 180,E1 3771.262,E2 3771.262} C_VEL
LIN {X 0,Y 105.627,Z 968.693,A -85,B 0,C 180,E1 3767.424,E2 3767.424} C_VEL
LIN {X 0,Y 87.379,Z 976.468,A -85,B 0,C 180,E1 3761.748,E2 3761.748} C_VEL
LIN {X 0,Y 69.614,Z 982.569,A -85,B 0,C 180,E1 3752.926,E2 3752.926} C_VEL
LIN {X 0,Y 54.305,Z 986.765,A -85,B 0,C 180,E1 3739.007,E2 3739.007} C_VEL
LIN {X 0,Y 44.072,Z 989.123,A -85,B 0,C 180,E1 3718.445,E2 3718.445} C_VEL
LIN {X 0,Y 40.629,Z 989.846,A -85,B 0,C 180,E1 3697.06,E2 3697.06} C_VEL
LIN {X 0,Y 40.802,Z 989.815,A -85,B 0,C 180,E1 3680.115,E2 3680.115} C_VEL
LIN {X 0,Y 45.625,Z 988.807,A -85,B 0,C 180,E1 3656.771,E2 3656.771} C_VEL
LIN {X 0,Y 56.921,Z 986.218,A -85,B 0,C 180,E1 3637.762,E2 3637.762} C_VEL
LIN {X 0,Y 72.841,Z 981.668,A -85,B 0,C 180,E1 3624.974,E2 3624.974} C_VEL
LIN {X 0,Y 61.094,Z 985.041,A -85,B 0,C 180,E1 3592.478,E2 3592.478} C_VEL
LIN {X 0,Y 64.444,Z 986.806,A -85,B 0,C 180,E1 3573.696,E2 3573.696} C_VEL
LIN {X 0,Y 49.952,Z 991.008,A -85,B 0,C 180,E1 3557.792,E2 3557.792} C_VEL
LIN {X 0,Y 41.488,Z 993.389,A -85,B 0,C 180,E1 3533.687,E2 3533.687} C_VEL
LIN {X 0,Y 40.545,Z 994.107,A -85,B 0,C 180,E1 3511.421,E2 3511.421} C_VEL
LIN {X 0,Y 40.409,Z 993.862,A -85,B 0,C 180,E1 3497.141,E2 3497.141} C_VEL
LIN {X 0,Y 45.723,Z 992.108,A -85,B 0,C 180,E1 3470.651,E2 3470.651} C_VEL
LIN {X 0,Y 58.512,Z 988.509,A -85,B 0,C 180,E1 3451.316,E2 3451.316} C_VEL
LIN {X 0,Y 74.466,Z 983.355,A -85,B 0,C 180,E1 3439.979,E2 3439.979} C_VEL
LIN {X 0,Y 92.265,Z 976.409,A -85,B 0,C 180,E1 3432.773,E2 3432.773} C_VEL
LIN {X 0,Y 111.043,Z 967.508,A -85,B 0,C 180,E1 3427.936,E2 3427.936} C_VEL
LIN {X 0,Y 129.411,Z 957.006,A -85,B 0,C 180,E1 3424.695,E2 3424.695} C_VEL
LIN {X 0,Y 147.103,Z 944.958,A -85,B 0,C 180,E1 3422.399,E2 3422.399} C_VEL
LIN {X 0,Y 162.988,Z 932.234,A -85,B 0,C 180,E1 3420.813,E2 3420.813} C_VEL
LIN {X 0,Y 178.975,Z 917.233,A -85,B 0,C 180,E1 3419.544,E2 3419.544} C_VEL
LIN {X 0,Y 184.473,Z 911.489,A -85,B 0,C 180,E1 3419.17,E2 3419.17} C_VEL
LIN {X 0,Y 187.871,Z 912.843,A -85,B 0,C 180,E1 3418.952,E2 3418.952} C_VEL
LIN {X 0,Y 187.871,Z 950.311,A -85,B 0,C 180,E1 3418.952,E2 3418.952} C_VEL
LIN {X 0,Y 158.026,Z 950.311,A -85,B 0,C 180,E1 3418.991,E2 3418.991} C_VEL
LIN {X 0,Y 156.026,Z 948.311,A -85,B 0,C 180,E1 3418.994,E2 3418.994} C_VEL
LIN {X 0,Y 156.026,Z 941.65,A -85,B 0,C 180,E1 3418.994,E2 3418.994} C_VEL
LIN {X 0,Y 152.947,Z 940.037,A -85,B 0,C 180,E1 3418.696,E2 3418.696} C_VEL
LIN {X 0,Y 135.193,Z 952.325,A -85,B 0,C 180,E1 3416.753,E2 3416.753} C_VEL
LIN {X 0,Y 117.569,Z 962.532,A -85,B 0,C 180,E1 3414.253,E2 3414.253} C_VEL
LIN {X 0,Y 99.28,Z 971.311,A -85,B 0,C 180,E1 3410.722,E2 3410.722} C_VEL
LIN {X 0,Y 80.584,Z 978.58,A -85,B 0,C 180,E1 3405.406,E2 3405.406} C_VEL
LIN {X 0,Y 62.051,Z 984.201,A -85,B 0,C 180,E1 3396.692,E2 3396.692} C_VEL
LIN {X 0,Y 45.836,Z 987.933,A -85,B 0,C 180,E1 3381.738,E2 3381.738} C_VEL
LIN {X 0,Y 35.179,Z 989.844,A -85,B 0,C 180,E1 3357.039,E2 3357.039} C_VEL
LIN {X 0,Y 32.486,Z 990.36,A -85,B 0,C 180,E1 3329.991,E2 3329.991} C_VEL
LIN {X 0,Y 35.169,Z 989.866,A -85,B 0,C 180,E1 3302.933,E2 3302.933} C_VEL
LIN {X 0,Y 45.816,Z 987.984,A -85,B 0,C 180,E1 3278.209,E2 3278.209} C_VEL
LIN {X 0,Y 62.147,Z 984.244,A -85,B 0,C 180,E1 3263.142,E2 3263.142} C_VEL
LIN {X 0,Y 53.332,Z 986.848,A -85,B 0,C 180,E1 3231.376,E2 3231.376} C_VEL
LIN {X 0,Y 55.401,Z 987.954,A -85,B 0,C 180,E1 3216.608,E2 3216.608} C_VEL
LIN {X 0,Y 39.753,Z 991.717,A -85,B 0,C 180,E1 3196.848,E2 3196.848} C_VEL
LIN {X 0,Y 32.567,Z 993.451,A -85,B 0,C 180,E1 3166.05,E2 3166.05} C_VEL
LIN {X 0,Y 32.591,Z 993.711,A -85,B 0,C 180,E1 3150.009,E2 3150.009} C_VEL
LIN {X 0,Y 34.256,Z 992.924,A -85,B 0,C 180,E1 3120.262,E2 3120.262} C_VEL
LIN {X 0,Y 45.514,Z 990.37,A -85,B 0,C 180,E1 3093.418,E2 3093.418} C_VEL
LIN {X 0,Y 62.155,Z 986.025,A -85,B 0,C 180,E1 3078.766,E2 3078.766} C_VEL
LIN {X 0,Y 80.383,Z 980.054,A -85,B 0,C 180,E1 3070.707,E2 3070.707} C_VEL
LIN {X 0,Y 99.472,Z 972.24,A -85,B 0,C 180,E1 3065.695,E2 3065.695} C_VEL
LIN {X 0,Y 118.499,Z 962.67,A -85,B 0,C 180,E1 3062.417,E2 3062.417} C_VEL
LIN {X 0,Y 135.977,Z 952.12,A -85,B 0,C 180,E1 3060.274,E2 3060.274} C_VEL
LIN {X 0,Y 152.947,Z 940.037,A -85,B 0,C 180,E1 3058.696,E2 3058.696} C_VEL
LIN {X 0,Y 156.084,Z 941.632,A -85,B 0,C 180,E1 3058.449,E2 3058.449} C_VEL
LIN {X 0,Y 156.084,Z 971.987,A -85,B 0,C 180,E1 3058.449,E2 3058.449} C_VEL
LIN {X 0,Y 123.426,Z 971.987,A -85,B 0,C 180,E1 3058.753,E2 3058.753} C_VEL
LIN {X 0,Y 121.426,Z 969.987,A -85,B 0,C 180,E1 3058.777,E2 3058.777} C_VEL
LIN {X 0,Y 121.426,Z 963.934,A -85,B 0,C 180,E1 3058.777,E2 3058.777} C_VEL
LIN {X 0,Y 118.655,Z 962.134,A -85,B 0,C 180,E1 3058.417,E2 3058.417} C_VEL
LIN {X 0,Y 99.278,Z 971.337,A -85,B 0,C 180,E1 3055.568,E2 3055.568} C_VEL
LIN {X 0,Y 78.929,Z 978.998,A -85,B 0,C 180,E1 3051.122,E2 3051.122} C_VEL
LIN {X 0,Y 59.31,Z 984.62,A -85,B 0,C 180,E1 3043.91,E2 3043.91} C_VEL
LIN {X 0,Y 41.318,Z 988.35,A -85,B 0,C 180,E1 3030.58,E2 3030.58} C_VEL
LIN {X 0,Y 28.256,Z 990.259,A -85,B 0,C 180,E1 3004.47,E2 3004.47} C_VEL
LIN {X 0,Y 24.496,Z 990.771,A -85,B 0,C 180,E1 2969.988,E2 2969.988} C_VEL
LIN {X 0,Y 28.247,Z 990.28,A -85,B 0,C 180,E1 2935.491,E2 2935.491} C_VEL
LIN {X 0,Y 41.303,Z 988.4,A -85,B 0,C 180,E1 2909.353,E2 2909.353} C_VEL
LIN {X 0,Y 51.676,Z 986.395,A -85,B 0,C 180,E1 2900.384,E2 2900.384} C_VEL
LIN {X 0,Y 45.432,Z 988.312,A -85,B 0,C 180,E1 2872.414,E2 2872.414} C_VEL
LIN {X 0,Y 46.315,Z 989.024,A -85,B 0,C 180,E1 2860.424,E2 2860.424} C_VEL
LIN {X 0,Y 30.692,Z 992.039,A -85,B 0,C 180,E1 2838.543,E2 2838.543} C_VEL
LIN {X 0,Y 24.365,Z 993.19,A -85,B 0,C 180,E1 2799.46,E2 2799.46} C_VEL
LIN {X 0,Y 24.471,Z 993.273,A -85,B 0,C 180,E1 2787.671,E2 2787.671} C_VEL
LIN {X 0,Y 27.939,Z 992.425,A -85,B 0,C 180,E1 2749.91,E2 2749.91} C_VEL
LIN {X 0,Y 42.379,Z 989.775,A -85,B 0,C 180,E1 2723.072,E2 2723.072} C_VEL
LIN {X 0,Y 61.072,Z 985.298,A -85,B 0,C 180,E1 2710.819,E2 2710.819} C_VEL
LIN {X 0,Y 80.242,Z 979.265,A -85,B 0,C 180,E1 2704.598,E2 2704.598} C_VEL
LIN {X 0,Y 99.99,Z 971.368,A -85,B 0,C 180,E1 2700.79,E2 2700.79} C_VEL
LIN {X 0,Y 118.655,Z 962.134,A -85,B 0,C 180,E1 2698.417,E2 2698.417} C_VEL
LIN {X 0,Y 121.498,Z 963.916,A -85,B 0,C 180,E1 2698.126,E2 2698.126} C_VEL
LIN {X 0,Y 121.498,Z 987.108,A -85,B 0,C 180,E1 2698.126,E2 2698.126} C_VEL
LIN {X 0,Y 88.482,Z 987.108,A -85,B 0,C 180,E1 2697.757,E2 2697.757} C_VEL
LIN {X 0,Y 86.483,Z 985.108,A -85,B 0,C 180,E1 2697.725,E2 2697.725} C_VEL
LIN {X 0,Y 86.483,Z 979.323,A -85,B 0,C 180,E1 2697.725,E2 2697.725} C_VEL
LIN {X 0,Y 83.874,Z 977.438,A -85,B 0,C 180,E1 2698.099,E2 2698.099} C_VEL
LIN {X 0,Y 63.034,Z 984.075,A -85,B 0,C 180,E1 2702.237,E2 2702.237} C_VEL
LIN {X 0,Y 43.623,Z 988.665,A -85,B 0,C 180,E1 2709.786,E2 2709.786} C_VEL
LIN {X 0,Y 25.214,Z 991.688,A -85,B 0,C 180,E1 2729.284,E2 2729.284} C_VEL
LIN {X 0,Y 16.362,Z 992.797,A -85,B 0,C 180,E1 2779.456,E2 2779.456} C_VEL
LIN {X 0,Y 16.433,Z 992.865,A -85,B 0,C 180,E1 2793.507,E2 2793.507} C_VEL
LIN {X 0,Y 23.064,Z 991.941,A -85,B 0,C 180,E1 2845.701,E2 2845.701} C_VEL
LIN {X 0,Y 37.826,Z 989.764,A -85,B 0,C 180,E1 2866.63,E2 2866.63} C_VEL
LIN {X 0,Y 40.847,Z 988.342,A -85,B 0,C 180,E1 2896.492,E2 2896.492} C_VEL
LIN {X 0,Y 23.203,Z 990.591,A -85,B 0,C 180,E1 2920.274,E2 2920.274} C_VEL
LIN {X 0,Y 16.577,Z 991.15,A -85,B 0,C 180,E1 2963.053,E2 2963.053} C_VEL
LIN {X 0,Y 19.764,Z 990.921,A -85,B 0,C 180,E1 3007.359,E2 3007.359} C_VEL
LIN {X 0,Y 34.483,Z 989.283,A -85,B 0,C 180,E1 3038.081,E2 3038.081} C_VEL
LIN {X 0,Y 52.81,Z 986.052,A -85,B 0,C 180,E1 3049.876,E2 3049.876} C_VEL
LIN {X 0,Y 73.162,Z 980.876,A -85,B 0,C 180,E1 3056.009,E2 3056.009} C_VEL
LIN {X 0,Y 83.874,Z 977.438,A -85,B 0,C 180,E1 3058.099,E2 3058.099} C_VEL
LIN {X 0,Y 73.721,Z 980.861,A -85,B 0,C 180,E1 3059.027,E2 3059.027} C_VEL
LIN {X 0,Y 56.546,Z 985.528,A -85,B 0,C 180,E1 3058.994,E2 3058.994} C_VEL
LIN {X 0,Y 42.189,Z 988.397,A -85,B 0,C 180,E1 3059.646,E2 3059.646} C_VEL
LIN {X 0,Y 36.228,Z 989.402,A -85,B 0,C 180,E1 3061.3,E2 3061.3} C_VEL
LIN {X 0,Y 16.897,Z 991.74,A -85,B 0,C 180,E1 3078.832,E2 3078.832} C_VEL
LIN {X 0,Y 8.457,Z 992.468,A -85,B 0,C 180,E1 3150.036,E2 3150.036} C_VEL
LIN {X 0,Y 18.889,Z 991.586,A -85,B 0,C 180,E1 3224.658,E2 3224.658} C_VEL
LIN {X 0,Y 29.574,Z 990.383,A -85,B 0,C 180,E1 3235.51,E2 3235.51} C_VEL
LIN {X 0,Y 30.779,Z 989.906,A -85,B 0,C 180,E1 3249.351,E2 3249.351} C_VEL
LIN {X 0,Y 13.47,Z 991.394,A -85,B 0,C 180,E1 3275.222,E2 3275.222} C_VEL
LIN {X 0,Y 8.696,Z 991.555,A -85,B 0,C 180,E1 3343.258,E2 3343.258} C_VEL
LIN {X 0,Y 19.279,Z 990.966,A -85,B 0,C 180,E1 3398.947,E2 3398.947} C_VEL
LIN {X 0,Y 39.153,Z 988.734,A -85,B 0,C 180,E1 3414.752,E2 3414.752} C_VEL
LIN {X 0,Y 47.577,Z 987.346,A -85,B 0,C 180,E1 3417.685,E2 3417.685} C_VEL
LIN {X 0,Y 36.228,Z 989.402,A -85,B 0,C 180,E1 3421.3,E2 3421.3} C_VEL
LIN {X 0,Y 28.345,Z 990.55,A -85,B 0,C 180,E1 3423.548,E2 3423.548} C_VEL
LIN {X 0,Y 16.201,Z 991.623,A -85,B 0,C 180,E1 3423.176,E2 3423.176} C_VEL
LIN {X 0,Y 1.673,Z 992.014,A -85,B 0,C 180,E1 3402.244,E2 3402.244} C_VEL
LIN {X 0,Y 0.904,Z 991.997,A -85,B 0,C 180,E1 3273.974,E2 3273.974} C_VEL
LIN {X 0,Y 4.015,Z 991.938,A -85,B 0,C 180,E1 3244.029,E2 3244.029} C_VEL
LIN {X 0,Y 0.378,Z 992.052,A -85,B 0,C 180,E1 3150.807,E2 3150.807} C_VEL
LIN {X 0,Y 4.011,Z 991.927,A -85,B 0,C 180,E1 3054.772,E2 3054.772} C_VEL
LIN {X 0,Y 0.904,Z 991.997,A -85,B 0,C 180,E1 2913.974,E2 2913.974} C_VEL
LIN {X 0,Y 2.809,Z 993.997,A -85,B 0,C 180,E1 2889.325,E2 2889.325} C_VEL
LIN {X 0,Y 2.809,Z 1028,A -85,B 0,C 180,E1 2889.325,E2 2889.325} C_VEL
LIN {X 0,Y 2.809,Z 1028,A -85,B 0,C 180,E1 2889.325,E2 2889.325}

QRS_NEXT_CUT()

QRS_NEXT()
QRS_HOME()

END
